{attribute 'qualified_only'}
VAR_GLOBAL
	// Rezept-Control-Words
	RZCW_R1				AT%Q*	:RezeptControlWord;				// Schnittstelle zur OPC UA Schnittstelle - Reaktor 1
END_VAR

(* stored: Version 1.1.0.1, ProductVersion 3.1.4024.12
   GVL GVL_OPC_UA: Id {13cb8d73-1df7-470b-8c80-ab1505072c03} *)
